(* CoDeSys 2.3.9.62 project: CruceMoviles.pro *)
(* Libraries: Standard.lib 2.6.14 11:37:46 *)

(* Global variable list: Global_Variables *)
VAR_GLOBAL

      (*Entradas*)
      M1:BOOL;
      M2:BOOL;

	A1:BOOL;
	B1:BOOL;
       C1: BOOL;
       D1:BOOL;

	A2:BOOL;
	B2:BOOL;
      C2: BOOL;
       D2:BOOL;

       (* Salidas *)
	MOTOR_BA1:BOOL;
	MOTOR_FO1:BOOL;

       MOTOR_BA2:BOOL;
	MOTOR_FO2:BOOL;

      Carga1:BOOL;
      Carga2:BOOL;


      (* Variables del simulador *)
	Vel:INT:=1;
	Vel2:INT:=1;


END_VAR

(* POU PLC_PRG, ST *)
PROGRAM PLC_PRG
VAR
END_VAR
SimVehiculo;
SimVehiculo2;
Automatismo;
END_PROGRAM

(* POU SimVehiculo, ST *)
PROGRAM SimVehiculo
VAR
	PosX: INT;
END_VAR
A1:=FALSE;
B1:=FALSE;
C1:=FALSE;
D1:=FALSE;


IF MOTOR_FO1=TRUE THEN

     PosX:=PosX+Vel;

END_IF

IF MOTOR_BA1=TRUE THEN

     PosX:=PosX-Vel;

END_IF


IF PosX<=0 THEN
   A1:=TRUE;
END_IF

IF PosX>=129 AND   PosX<=199 THEN
   B1:=TRUE;
END_IF

IF PosX>=220 AND   PosX<=288 THEN
   C1:=TRUE;
END_IF

IF PosX>=438 THEN
  D1:=TRUE;
END_IF
END_PROGRAM

(* POU SimVehiculo2, ST *)
PROGRAM SimVehiculo2
VAR
	PosY2: INT;
END_VAR
A2:=FALSE;
B2:=FALSE;
C2:=FALSE;
D2:=FALSE;


IF MOTOR_FO2=TRUE THEN

     PosY2:=PosY2-Vel2;

END_IF

IF MOTOR_BA2=TRUE THEN

     PosY2:=PosY2+Vel2;

END_IF


IF PosY2>=0 THEN
   A2:=TRUE;
END_IF

IF PosY2<=-70 AND PosY2>=-142 THEN
  B2:=TRUE;
END_IF

IF PosY2<=-151 AND PosY2>=-220 THEN
  C2:=TRUE;
END_IF

IF PosY2<=-302  THEN
  D2:=TRUE;
END_IF
END_PROGRAM

(* POU Automatismo, LD *)
PROGRAM Automatismo
VAR
	Carrito1:Carrito;
	Carrito2: Carrito;
END_VAR
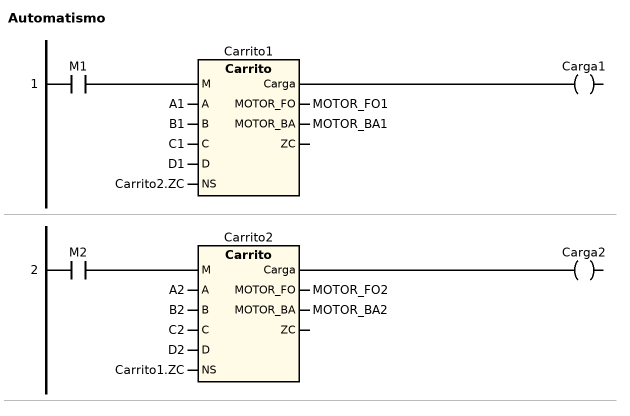
_LD_ (* Ladder Diagram *)
NETWORK 1
	[M1] - Carrito1:Carrito(M: *, A: A1, B: B1, C: C1, D: D1, NS: Carrito2.ZC, MOTOR_FO => MOTOR_FO1, MOTOR_BA => MOTOR_BA1) --- (Carga1)
NETWORK 2
	[M2] - Carrito2:Carrito(M: *, A: A2, B: B2, C: C2, D: D2, NS: Carrito1.ZC, MOTOR_FO => MOTOR_FO2, MOTOR_BA => MOTOR_BA2) --- (Carga2)
_END_LD_
(* the same logic as Structured Text *)
(* Network 1 *)
Carrito1(M := M1, A := A1, B := B1, C := C1, D := D1, NS := Carrito2.ZC);
MOTOR_FO1 := Carrito1.MOTOR_FO;
MOTOR_BA1 := Carrito1.MOTOR_BA;
Carga1 := Carrito1.Carga;
(* Network 2 *)
Carrito2(M := M2, A := A2, B := B2, C := C2, D := D2, NS := Carrito1.ZC);
MOTOR_FO2 := Carrito2.MOTOR_FO;
MOTOR_BA2 := Carrito2.MOTOR_BA;
Carga2 := Carrito2.Carga;
END_PROGRAM

(* POU Carrito, LD *)
FUNCTION_BLOCK Carrito
VAR_INPUT
	M:BOOL;
	A:BOOL;
	B:BOOL;
	C:BOOL;
	D:BOOL;
	NS:BOOL;(*Abreviatura de no es seguro*)
END_VAR
VAR_OUTPUT
	Carga:BOOL;
	MOTOR_FO:BOOL;
	MOTOR_BA:BOOL;
	ZC:BOOL;(* true si está en la zona crítica*)
END_VAR
VAR

	RC: R_TRIG;
	RB: R_TRIG;
	FC: F_TRIG;
	FB: F_TRIG;
	FCarga: F_TRIG;
	Continua: BOOL;

	ContaVueltas: CTD;
	NoContinua: BOOL;
	MSeguro: BOOL;
	TempCarga: TP;
END_VAR
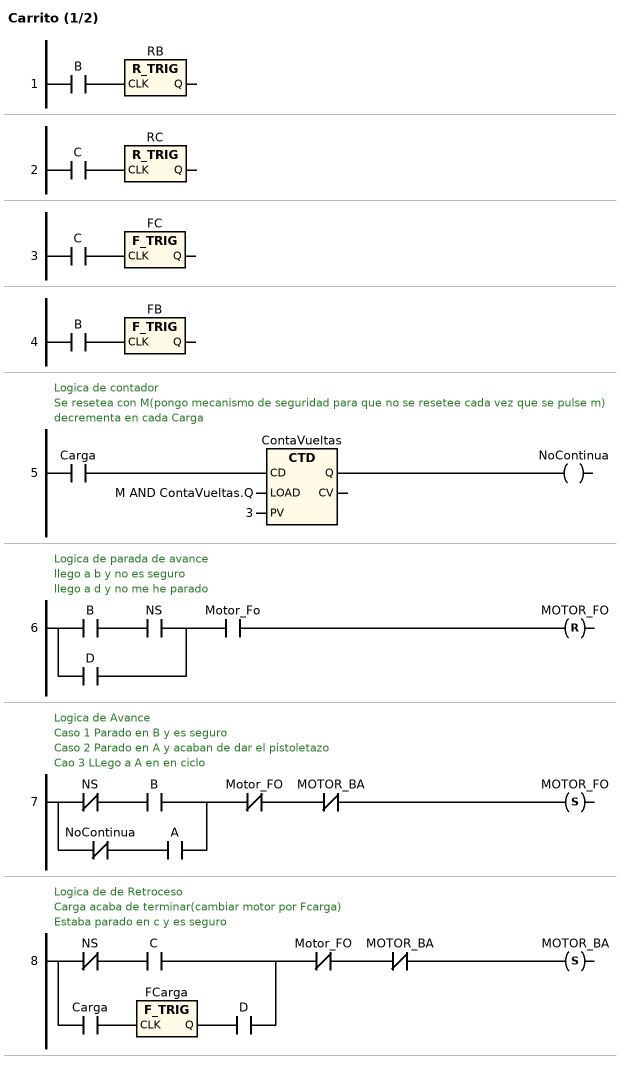
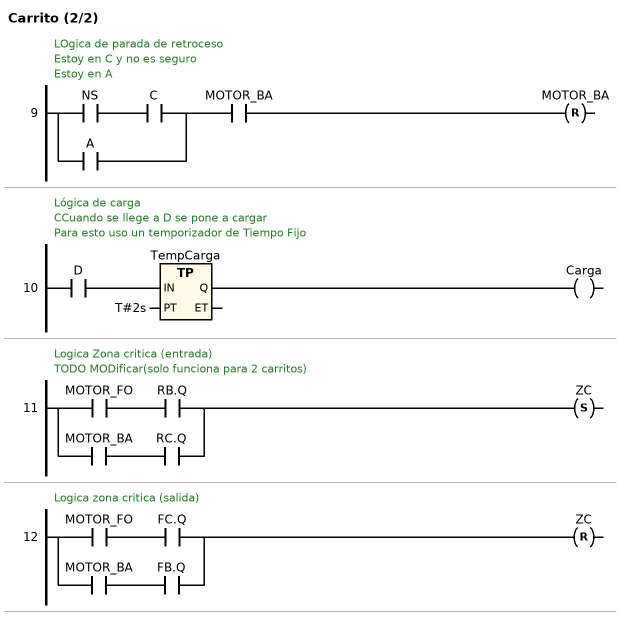
_LD_ (* Ladder Diagram *)
NETWORK 1
	[B] - RB:R_TRIG(CLK: *)
NETWORK 2
	[C] - RC:R_TRIG(CLK: *)
NETWORK 3
	[C] - FC:F_TRIG(CLK: *)
NETWORK 4
	[B] - FB:F_TRIG(CLK: *)
NETWORK 5 (* Logica de contador / Se resetea con M(pongo mecanismo de seguridad para que no se resetee cada vez que se pulse m) / decrementa en cada Carga *)
	[Carga] - ContaVueltas:CTD(CD: *, LOAD: M AND ContaVueltas.Q, PV: 3) --- (NoContinua)
NETWORK 6 (* Logica de parada de avance / llego a b y no es seguro / llego a d y no me he parado *)
	{ [B] - [NS] | [D] } - [Motor_Fo] --- (R MOTOR_FO)
NETWORK 7 (* Logica de Avance / Caso 1 Parado en B y es seguro / Caso 2 Parado en A y acaban de dar el pistoletazo / Cao 3 LLego a A en en ciclo *)
	{ [/NS] - [B] | [/NoContinua] - [A] } - [/Motor_FO] - [/MOTOR_BA] --- (S MOTOR_FO)
NETWORK 8 (* Logica de de Retroceso / Carga acaba de terminar(cambiar motor por Fcarga) / Estaba parado en c y es seguro *)
	{ [/NS] - [C] | [Carga] - FCarga:F_TRIG(CLK: *) - [D] } - [/Motor_FO] - [/MOTOR_BA] --- (S MOTOR_BA)
NETWORK 9 (* LOgica de parada de retroceso / Estoy en C y no es seguro / Estoy en A *)
	{ [NS] - [C] | [A] } - [MOTOR_BA] --- (R MOTOR_BA)
NETWORK 10 (* Lógica de carga / CCuando se llege a D se pone a cargar / Para esto uso un temporizador de Tiempo Fijo *)
	[D] - TempCarga:TP(IN: *, PT: T#2s) --- (Carga)
NETWORK 11 (* Logica Zona critica (entrada) / TODO MODificar(solo funciona para 2 carritos) *)
	{ [MOTOR_FO] - [RB.Q] | [MOTOR_BA] - [RC.Q] } --- (S ZC)
NETWORK 12 (* Logica zona critica (salida) *)
	{ [MOTOR_FO] - [FC.Q] | [MOTOR_BA] - [FB.Q] } --- (R ZC)
_END_LD_
(* the same logic as Structured Text *)
(* Network 1 *)
RB(CLK := B);
(* Network 2 *)
RC(CLK := C);
(* Network 3 *)
FC(CLK := C);
(* Network 4 *)
FB(CLK := B);
(* Network 5: Logica de contador / Se resetea con M(pongo mecanismo de seguridad para que no se resetee cada vez que se pulse m) / decrementa en cada Carga *)
ContaVueltas(CD := Carga, LOAD := M AND ContaVueltas.Q, PV := 3);
NoContinua := ContaVueltas.Q;
(* Network 6: Logica de parada de avance / llego a b y no es seguro / llego a d y no me he parado *)
IF (B AND NS OR D) AND Motor_Fo THEN MOTOR_FO := FALSE; END_IF;
(* Network 7: Logica de Avance / Caso 1 Parado en B y es seguro / Caso 2 Parado en A y acaban de dar el pistoletazo / Cao 3 LLego a A en en ciclo *)
IF (NOT NS AND B OR NOT NoContinua AND A) AND NOT Motor_FO AND NOT MOTOR_BA THEN MOTOR_FO := TRUE; END_IF;
(* Network 8: Logica de de Retroceso / Carga acaba de terminar(cambiar motor por Fcarga) / Estaba parado en c y es seguro *)
FCarga(CLK := Carga);
IF (NOT NS AND C OR FCarga.Q AND D) AND NOT Motor_FO AND NOT MOTOR_BA THEN MOTOR_BA := TRUE; END_IF;
(* Network 9: LOgica de parada de retroceso / Estoy en C y no es seguro / Estoy en A *)
IF (NS AND C OR A) AND MOTOR_BA THEN MOTOR_BA := FALSE; END_IF;
(* Network 10: Lógica de carga / CCuando se llege a D se pone a cargar / Para esto uso un temporizador de Tiempo Fijo *)
TempCarga(IN := D, PT := T#2s);
Carga := TempCarga.Q;
(* Network 11: Logica Zona critica (entrada) / TODO MODificar(solo funciona para 2 carritos) *)
IF MOTOR_FO AND RB.Q OR MOTOR_BA AND RC.Q THEN ZC := TRUE; END_IF;
(* Network 12: Logica zona critica (salida) *)
IF MOTOR_FO AND FC.Q OR MOTOR_BA AND FB.Q THEN ZC := FALSE; END_IF;
END_FUNCTION_BLOCK

(* Visualisation Vehiculo
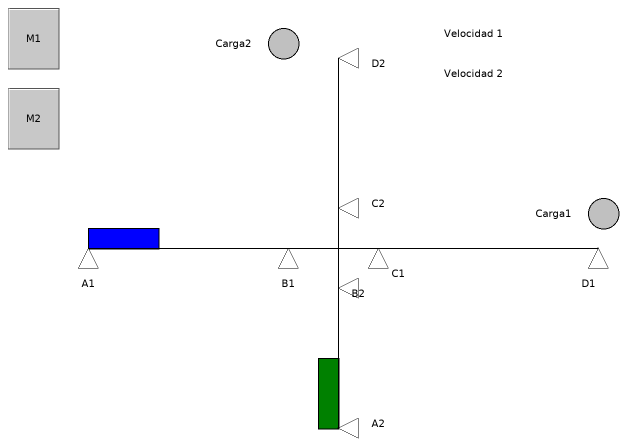
rectangle at (120,230)-(191,251): x offset SimVehiculo.PosX
polygon at (110,250)-(130,270): alarm colour if .A1
polygon at (620,250)-(640,270): alarm colour if .D1
button at (40,10)-(91,71): text "M1"; taps M1
rectangle at (350,360)-(371,431): y offset SimVehiculo2.PosY2
polygon at (370,420)-(390,440): alarm colour if .A2
rectangle at (450,20)-(561,51): text "Velocidad 1"
rectangle at (450,60)-(561,91): text "Velocidad 2"
polygon at (370,50)-(390,70): alarm colour if .D2
polygon at (310,250)-(330,270): alarm colour if .B1
polygon at (400,250)-(420,270): alarm colour if .C1
polygon at (370,280)-(390,300): alarm colour if .B2
polygon at (370,200)-(390,220): alarm colour if .C2
ellipse at (620,200)-(651,231): alarm colour if Carga1
rectangle at (530,200)-(641,231): text "Carga1"
ellipse at (300,30)-(331,61): alarm colour if Carga2
rectangle at (210,30)-(321,61): text "Carga2"
rectangle at (100,270)-(141,301): text "A1"
rectangle at (300,270)-(341,301): text "B1"
rectangle at (410,260)-(451,291): text "C1"
rectangle at (600,270)-(641,301): text "D1"
rectangle at (390,410)-(431,441): text "A2"
rectangle at (370,280)-(411,311): text "B2"
rectangle at (390,190)-(431,221): text "C2"
rectangle at (390,50)-(431,81): text "D2"
button at (40,90)-(91,151): text "M2"; taps M2
2 more shapes without text or variables
2 elements of other kinds (tables, trends, ...) not read
*)
